// TIA Portal V21 export
DATA_BLOCK "CipRe"   // DB42
{ S7_Optimized_Access := 'TRUE' }
// stored: MemoryReserve 100
   VAR
      CipLinePrintText : Array[0..20] of String;
   END_VAR
BEGIN
   CipLinePrintText[1] := 'PRE RINSE CYCLE - RINSING ON STARTED';
   CipLinePrintText[2] := 'PRE RINSE CYCLE - DRAIN ON STARTED';
   CipLinePrintText[3] := 'PRE RINSE CYCLE - SYSTEM DRAIN STARTED';
   CipLinePrintText[4] := 'PRE RINSE CYCLE - AIR PURGING STARTED';
   CipLinePrintText[5] := 'FILLING CYCLE - FILLING ON STARTED';
   CipLinePrintText[6] := 'FILLING CYCLE - MIXING ON STARTED';
   CipLinePrintText[7] := 'FILLING CYCLE - DRAIN ON STARTED';
   CipLinePrintText[8] := 'FILLING CYCLE - SYSTEM DRAIN STARTED';
   CipLinePrintText[9] := 'FILLING CYCLE - AIR PURGING ON STARTED';
   CipLinePrintText[10] := 'WAITING FOR ACKNOWLEDGE';
   CipLinePrintText[11] := 'CYCLE PAUSED';
   CipLinePrintText[12] := 'CIP CYCLE OVER';
   CipLinePrintText[13] := 'CYCLE RESETED';
   CipLinePrintText[14] := 'FILLING CYCLE - RECIRCULATION STARTED';
   CipLinePrintText[15] := 'FINAL RINSE CYCLE - FILLING ON STARTED';
   CipLinePrintText[16] := 'FINAL RINSE CYCLE - MIXING ON STARTED';
   CipLinePrintText[17] := 'FINAL RINSE CYCLE - DRAIN ON STARTED';
   CipLinePrintText[18] := 'FINAL RINSE CYCLE - SYSTEM DRAIN STARTED';
   CipLinePrintText[19] := 'FINAL RINSE CYCLE - AIR PURGING ON STARTED';
   CipLinePrintText[20] := 'FINAL RINSE CYCLE - RECIRCULATION STARTED';
END_DATA_BLOCK
